Fanuc TP program (LS listing): _CELLMON.LS

/PROG  _CELLMON	  Cond
/ATTR
OWNER		= MNEDITOR;
COMMENT		= "Fanuc Alarm Mon";
PROG_SIZE	= 330;
CREATE		= DATE 21-03-19  TIME 11:14:44;
MODIFIED	= DATE 21-03-19  TIME 11:14:44;
FILE_NAME	= ;
VERSION		= 0;
LINE_COUNT	= 7;
MEMORY_SIZE	= 730;
PROTECT		= READ_WRITE;
TCD:  STACK_SIZE	= 0,
      TASK_PRIORITY	= 50,
      TIME_SLICE	= 0,
      BUSY_LAMP_OFF	= 0,
      ABORT_REQUEST	= 0,
      PAUSE_REQUEST	= 7;
DEFAULT_GROUP	= *,*,*,*,*;
CONTROL_CODE	= 00000000 00000000;
/APPL
/MN
   1:  WHEN ERR_NUM=15018,CALL _FLTPNR ;
   2:  WHEN ERR_NUM=11050,CALL _FLTCOL ;
   3:  WHEN ERR_NUM=15017,CALL _FLTLIM ;
   4:  WHEN ERR_NUM=11045,CALL _FLTHCAL ;
   5:  WHEN ERR_NUM=11046,CALL _FLTOVC ;
   6:  WHEN ERR_NUM=11023,CALL _FLTSEE ;
   7:  WHEN ERR_NUM=11024,CALL _FLTMEE ;
/POS
/END
